PROGRAM P90_Interlock
VAR_INPUT
	bRecipeRunning 		: BOOL;
	RecipeStopped 		: BOOL;
	ManualOperation 	: BOOL;
	bInductionHeaterMC	: BOOL;
	bThermalBathMC		: BOOL;
	bVacuumPumpMC 		: BOOL;
	bLineHeaterMC 		: BOOL; 
END_VAR
VAR_OUTPUT
	bRecipeStartAvailable	: BOOL;
	bReactorOpenEnable		: BOOL;
	bHeaterOnEnable			: BOOL;
	bPumpOnEnable			: BOOL;
	
	bDorOnEnable			: BOOL;
	bDorOffEnable			: BOOL;
	bOpenEnableTemp			: BOOL;
	bOpenEnablePress		: BOOL;	
	
	bPowerResetSwitch		: BOOL;
	bMainPowerMonitor		: BOOL;

	AlarmTrig				: BOOL;
	WarningTrig				: BOOL;
	bMaintKey				: BOOL;
	bGasStateProcess		: BOOL;
	bGasStateSource			: BOOL;
	bGasStateVent			: BOOL;
END_VAR	
VAR
	bPowerResetLED			: BOOL;
	bUPSMode				: BOOL;
	tAlarmDelay_A			: TIME; //아날로그 디바이스 지연시간
	tAlarmDelay_D			: TIME; //디지털 디바이스 지연시간
	
	fbDeviationCheck		:ARRAY[1..29] OF FB_DeviationCheck;
	wDeviceAlarmEnable		: DWORD;
	wDeviceWarningEnable	: DWORD;
	bDeviationAlarm			: BOOL;
	bDeviationWarning		: BOOL;
	wDeviationAlarm			: DWORD;
	wDeviationWarning		: DWORD;

	fbSensorLimitCheck		:ARRAY[1..4] OF FB_SensorLimitCheck;
	wLimitAlarmEnable		: DWORD;
	wLimitWarningEnable		: DWORD;
	bLimitAlarm				: BOOL;
	bLimitWarning			: BOOL;
	wLimitAlarm				: DWORD;
	wLimitWarning			: DWORD;
	
	fbFaultCheck			:ARRAY[1..6] OF FB_FaultCheck;
	wAlarmEnable			: DWORD;
	wWarningEnable			: DWORD;

	bFaultAlarm				: BOOL;
	bFaultWarning			: BOOL;
	wAlarm					: DWORD;
	wWarning				: DWORD;
		
	bAlarmEnable			: BOOL;
	bWarningEnable			: BOOL;
	bDeviceCurrentAlarmState	: BOOL;
	bDeviceCurrentWarningState 	: BOOL;
	fDeviceCurrentValue			: REAL;
	fDeviceAlarmTreshold		: REAL;
	fDeviceWarningTreshold		: REAL;
	
	i	: INT;
	j 	: INT;
	
END_VAR

(* Read from Device*)
//Interlock Variable Set
bMaintKey := GVL_IO.aDigitalInputIO[1].0;
bPowerResetSwitch := GVL_IO.aDigitalInputIO[1].1;
bMainPowerMonitor := GVL_IO.aDigitalInputIO[7].5;
bGasStateProcess := GVL_IO.aOutputSolValve[1].0 AND //HYD Carrier Change Valve
	GVL_IO.aOutputSolValve[1].1 AND //Main Carrier Change Valve
	GVL_IO.aOutputSolValve[1].2 AND //SiH4 Source Change Valve
	GVL_IO.aOutputSolValve[1].3 //NH3 Source Change Valve
	; //All False이면 Safety State
bGasStateSource := GVL_IO.aOutputSolValve[1].4 AND GVL_IO.aOutputSolValve[1].5 AND GVL_IO.aOutputSolValve[1].6 AND //Source #1
	GVL_IO.aOutputSolValve[1].7 AND GVL_IO.aOutputSolValve[1].8 AND GVL_IO.aOutputSolValve[1].9 AND //Source #2
	GVL_IO.aOutputSolValve[1].10 AND GVL_IO.aOutputSolValve[1].11 AND GVL_IO.aOutputSolValve[1].12 AND //Source #3
	GVL_IO.aOutputSolValve[1].13 AND GVL_IO.aOutputSolValve[1].14 AND GVL_IO.aOutputSolValve[1].15 AND //Source #4
	GVL_IO.aOutputSolValve[2].0 AND GVL_IO.aOutputSolValve[2].1 AND GVL_IO.aOutputSolValve[2].2 AND //Source #5
	GVL_IO.aOutputSolValve[2].3 AND GVL_IO.aOutputSolValve[2].4 AND GVL_IO.aOutputSolValve[2].6 //Source #6
	; //All False이면 Safety State
bGasStateVent := GVL_IO.aOutputSolValve[2].15;
GVL_IO.aInterlock[1].10 := bRecipeStartAvailable;
GVL_IO.aInterlock[1].11 := bReactorOpenEnable;
GVL_IO.aInterlock[1].12 := bHeaterOnEnable;
GVL_IO.aInterlock[1].13 := bPumpOnEnable;

//Sinal Tower Set
IF (bMaintKey = TRUE) THEN //bMaintKey 변경
	P92_Maintenance.nCaseSignalTower		:= 5; //Signal Tower White - Maintenance
ELSIF (bMaintKey = FALSE) AND MAIN.bOperationMode = FALSE THEN
	P92_Maintenance.nCaseSignalTower		:= 4; //Signal Tower Blue - Idle
END_IF

//알람 지연 시간 변환
tAlarmDelay_A := REAL_TO_TIME(GVL_IO.aInterlockSet[3]*1000); // UI Setting Analog Delay Time Value(Miliseconde)
tAlarmDelay_D := REAL_TO_TIME(GVL_IO.aInterlockSet[4]*1000);

//Controller Deviation Monitoring - MFC/EPC
IF (bMaintKey = FALSE) THEN
	FOR i := 1 TO 26 DO
		wDeviceAlarmEnable := SHR(GVL_IO.aInterlockEnable[2], (i+2)); //오늘쪽 쉬프트 연산
		wDeviceWarningEnable := SHR(GVL_IO.aInterlockEnable[3], (i+2));
		fbDeviationCheck[i](
			bAlarmEnable := wDeviceAlarmEnable.0,
			bWarningEnable := wDeviceWarningEnable.0,
			fCurrentValue := GVL_IO.aController_PV[i],
			fControlValue := GVL_IO.aController_CV[i],
			fMaxValue := GVL_IO.aMaxValueController[i],
			fAlarmTreshold := GVL_IO.aInterlockSet[1],
			fWarningTreshold := GVL_IO.aInterlockSet[2],
			tAlarmDelay := tAlarmDelay_A,
			bDeviationAlarm => bDeviationAlarm, //알람 출력
			bDeviationWarning => bDeviationWarning // 주의(Warning) 출력
			);
		IF bDeviationAlarm THEN		
			GVL_IO.aInterlock[1].0 := TRUE; //Alarm Trig
			P92_Maintenance.nCaseSignalTower := 1; // Signal Tower RED - Alarm
			wDeviationAlarm := ROR(GVL_IO.aInterlock[3], (i+2));
			wDeviationAlarm.0 := TRUE;
			GVL_IO.aInterlock[3] := ROL(wDeviationAlarm, (i+2));
		ELSE
			wDeviationAlarm := ROR(GVL_IO.aInterlock[3], (i+2));
			wDeviationAlarm.0 := FALSE;
			GVL_IO.aInterlock[3] := ROL(wDeviationAlarm, (i+2));	
		END_IF
		
		IF bDeviationWarning THEN
			GVL_IO.aInterlock[1].1 := TRUE; // Warning Trig
			P92_Maintenance.nCaseSignalTower := 2; // Signal Tower Yellow - Warning
			wDeviationWarning := ROR(GVL_IO.aInterlock[5], (i+2));
			wDeviationWarning.0 := TRUE;
			GVL_IO.aInterlock[5] := ROL(wDeviationWarning, (i+2));
		ELSE
			wDeviationWarning := ROR(GVL_IO.aInterlock[5], (i+2));
			wDeviationWarning.0 := FALSE;
			GVL_IO.aInterlock[5] := ROL(wDeviationWarning, (i+2));
		END_IF
	END_FOR
	//Controller Deviation Monitoring - Temp, Pressure, Rotation
	FOR i := 27 TO 29 DO
		wDeviceAlarmEnable := SHR(GVL_IO.aInterlockEnable[2], (i-27)); //오늘쪽 쉬프트 연산, -27은 어레이 변수 옵셋값
		wDeviceWarningEnable := SHR(GVL_IO.aInterlockEnable[3], (i-27));
		fbDeviationCheck[i](
			bAlarmEnable := wDeviceAlarmEnable.0,
			bWarningEnable := wDeviceWarningEnable.0,
			fCurrentValue := GVL_IO.aController_PV[i],
			fControlValue := GVL_IO.aController_CV[i],
			fMaxValue := GVL_IO.aMaxValueController[i],
			fAlarmTreshold := GVL_IO.aInterlockSet[1],
			fWarningTreshold := GVL_IO.aInterlockSet[2],
			tAlarmDelay := tAlarmDelay_A,
			bDeviationAlarm => bDeviationAlarm, //알람 출력
			bDeviationWarning => bDeviationWarning // 주의(Warning) 출력
			);
		IF bDeviationAlarm THEN		
			GVL_IO.aInterlock[1].0 := TRUE; //Alarm Trig
			P92_Maintenance.nCaseSignalTower := 1; // Signal Tower RED - Alarm
			wDeviationAlarm := ROR(GVL_IO.aInterlock[3], (i-27));
			wDeviationAlarm.0 := TRUE;
			GVL_IO.aInterlock[3] := ROL(wDeviationAlarm, (i-27));
		ELSE
			wDeviationAlarm := ROR(GVL_IO.aInterlock[3], (i-27));
			wDeviationAlarm.0 := FALSE;
			GVL_IO.aInterlock[3] := ROL(wDeviationAlarm, (i-27));
		END_IF
		
		IF bDeviationWarning THEN
			GVL_IO.aInterlock[1].1 := TRUE; // Warning Trig
			P92_Maintenance.nCaseSignalTower := 2; // Signal Tower Yellow - Warning
			wDeviationWarning := ROR(GVL_IO.aInterlock[5], (i-27));
			wDeviationWarning.0 := TRUE;
			GVL_IO.aInterlock[5] := ROL(wDeviationWarning, (i-27));
		ELSE
			wDeviationWarning := ROR(GVL_IO.aInterlock[5], (i-27));
			wDeviationWarning.0 := FALSE;
			GVL_IO.aInterlock[5] := ROL(wDeviationWarning, (i-27));
		END_IF	
	END_FOR
	//Gas Pressure Alarm N2, H2, NH3, SiH4
	FOR i := 1 TO 4 DO
		wLimitAlarmEnable := SHR(GVL_IO.aInterlockEnable[4], (i-1)); //오늘쪽 쉬프트 연산, 은 어레이 변수 옵셋값
		wLimitWarningEnable := SHR(GVL_IO.aInterlockEnable[5], (i-1));
		fbSensorLimitCheck[i](
			bAlarmEnable := wLimitAlarmEnable.0,
			bWarningEnable := wLimitWarningEnable.0,
			fCurrentValue := GVL_IO.aMonitoring_PV[(i+3)],
			fAlarmTreshold := GVL_IO.aInterlockSet[5],
			fWarningTreshold := GVL_IO.aInterlockSet[6],
			tAlarmDelay := tAlarmDelay_D,
			bLimitAlarm => bLimitAlarm, //알람 출력
			bLimitWarning => bLimitWarning //주의(Warning) 출력
			);	
		IF bLimitAlarm THEN		
			GVL_IO.aInterlock[1].0 := TRUE; //Alarm Trig
			P92_Maintenance.nCaseSignalTower := 1; // Signal Tower RED - Alarm
			//팝업 표시
			wLimitAlarm := ROR(GVL_IO.aInterlock[2], (i-1));
			wLimitAlarm.0 := TRUE;
			GVL_IO.aInterlock[2] := ROL(wLimitAlarm, (i-1));
			//대시보드 표시
			wLimitAlarm := ROR(GVL_IO.aInterlock[1], (i*2));
			wLimitAlarm.0 := TRUE;
			GVL_IO.aInterlock[1] := ROL(wLimitAlarm, (i*2));
		ELSE
			//팝업 표시
			wLimitAlarm := ROR(GVL_IO.aInterlock[2], (i-1));
			wLimitAlarm.0 := FALSE;
			GVL_IO.aInterlock[2] := ROL(wLimitAlarm, (i-1));
			//대시보드 표시
			wLimitAlarm := ROR(GVL_IO.aInterlock[1], (i*2));
			wLimitAlarm.0 := FALSE;
			GVL_IO.aInterlock[1] := ROL(wLimitAlarm, (i*2));
		END_IF
		
		IF bLimitWarning THEN		
			GVL_IO.aInterlock[1].1 := TRUE; //Warning Trig
			P92_Maintenance.nCaseSignalTower := 2; // Signal Tower YELLOW - Warning
			//팝업 표시
			wLimitWarning := ROR(GVL_IO.aInterlock[4], (i-1));
			wLimitWarning.0 := TRUE;
			GVL_IO.aInterlock[4] := ROL(wLimitWarning, (i-1));
			//대시보드 표시
			wLimitWarning := ROR(GVL_IO.aInterlock[1], (i*2)+1);
			wLimitWarning.0 := TRUE;
			GVL_IO.aInterlock[1] := ROL(wLimitWarning, (i*2)+1);
		ELSE
			//팝업 표시
			wLimitWarning := ROR(GVL_IO.aInterlock[4], (i-1));
			wLimitWarning.0 := FALSE;
			GVL_IO.aInterlock[4] := ROL(wLimitWarning, (i-1));
			//대시보드 표시
			wLimitWarning := ROR(GVL_IO.aInterlock[1], (i*2)+1);
			wLimitWarning.0 := FALSE;
			GVL_IO.aInterlock[1] := ROL(wLimitWarning, (i*2)+1);
		END_IF
	END_FOR
	
	//Cooling Water Over Temperature, Susceptor Over Temperature, Reactor Over Pressure
	FOR i := 1 TO 4 DO
		CASE i OF
			1: //CW Temperature High S/H
				bAlarmEnable := GVL_IO.aInterlockEnable[4].4;
				bWarningEnable := GVL_IO.aInterlockEnable[5].4;
				fDeviceCurrentValue := GVL_IO.aMonitoring_PV[8];
				fDeviceAlarmTreshold := GVL_IO.aInterlockSet[7];
				fDeviceWarningTreshold := GVL_IO.aInterlockSet[8];
			2: //CW Temperature High Coil
				bAlarmEnable := GVL_IO.aInterlockEnable[4].5;
				bWarningEnable := GVL_IO.aInterlockEnable[5].5;
				fDeviceCurrentValue := GVL_IO.aMonitoring_PV[9];
				fDeviceAlarmTreshold := GVL_IO.aInterlockSet[9];
				fDeviceWarningTreshold := GVL_IO.aInterlockSet[10];
			3: //Susceptor Over Temperature
				bAlarmEnable := GVL_IO.aInterlockEnable[4].6;
				bWarningEnable := GVL_IO.aInterlockEnable[5].6;
				fDeviceCurrentValue := GVL_IO.aController_PV[27];
				fDeviceAlarmTreshold := GVL_IO.aInterlockSet[11];
				fDeviceWarningTreshold := (GVL_IO.aInterlockSet[11] - 20.0); //20도 아래에서 Warning 발생				
			4: //Reactor Over Pressure Alarm
				bAlarmEnable := GVL_IO.aInterlockEnable[4].7;
				bWarningEnable := GVL_IO.aInterlockEnable[5].7;
				fDeviceCurrentValue := GVL_IO.aController_PV[28];
				fDeviceAlarmTreshold := GVL_IO.aInterlockSet[12];
				fDeviceWarningTreshold := (GVL_IO.aInterlockSet[12] - 50.0); //50Torr 아래에서 Warning 발생							
		END_CASE
		fbSensorLimitCheck[i](
			bAlarmEnable := bAlarmEnable,
			bWarningEnable := bWarningEnable,
			fCurrentValue := fDeviceCurrentValue,
			fAlarmTreshold := fDeviceAlarmTreshold,
			fWarningTreshold := fDeviceWarningTreshold,
			tAlarmDelay := tAlarmDelay_D,
			bLimitAlarm => bLimitAlarm, //알람 출력
			bLimitWarning => bLimitWarning //주의(Warning) 출력
			);
		IF bLimitAlarm THEN		
			GVL_IO.aInterlock[1].0 := TRUE; //Alarm Trig
			P92_Maintenance.nCaseSignalTower := 1; // Signal Tower RED - Alarm
			wDeviationAlarm := ROR(GVL_IO.aInterlock[2], (i+3));
			wDeviationAlarm.0 := TRUE;
			GVL_IO.aInterlock[2] := ROL(wDeviationAlarm, (i+3));
		ELSE
			wDeviationAlarm := ROR(GVL_IO.aInterlock[2], (i+3));
			wDeviationAlarm.0 := FALSE;
			GVL_IO.aInterlock[2] := ROL(wDeviationAlarm, (i+3));
		END_IF
		
		IF bDeviationWarning THEN
			GVL_IO.aInterlock[1].1 := TRUE; // Warning Trig
			P92_Maintenance.nCaseSignalTower := 2; // Signal Tower Yellow - Warning
			wDeviationWarning := ROR(GVL_IO.aInterlock[4], (i+3));
			wDeviationWarning.0 := TRUE;
			GVL_IO.aInterlock[4] := ROL(wDeviationWarning, (i+3));
		ELSE
			wDeviationWarning := ROR(GVL_IO.aInterlock[4], (i+3));
			wDeviationWarning.0 := FALSE;
			GVL_IO.aInterlock[4] := ROL(wDeviationWarning, (i+3));
		END_IF		
	END_FOR
	
	//Device Fault Check - Pneumatic, Heater, Pump, Motor, GC Door, RC Door
	FOR i := 1 TO 8 DO
		CASE i OF
			1: //CDA Alarm Switch (Pneumatic)
				bAlarmEnable := GVL_IO.aInterlockEnable[4].8;
				bWarningEnable := GVL_IO.aInterlockEnable[5].8;
				bDeviceCurrentAlarmState := GVL_IO.aInputState[1].4;
				bDeviceCurrentWarningState := GVL_IO.aInputState[1].4;
			2: //Cooling Water Switch
				bAlarmEnable := GVL_IO.aInterlockEnable[4].9;
				bWarningEnable := GVL_IO.aInterlockEnable[5].9;
				bDeviceCurrentAlarmState := GVL_IO.aInputState[1].5;
				bDeviceCurrentWarningState := GVL_IO.aInputState[1].5;
			3: //Induction Heater Fault
				bAlarmEnable := GVL_IO.aInterlockEnable[4].10;
				bWarningEnable := GVL_IO.aInterlockEnable[5].10;
				bDeviceCurrentAlarmState := GVL_IO.aInputState[1].8;
				bDeviceCurrentWarningState := GVL_IO.aInputState[1].8;
			4: //Rotatin Motor Fault
				bAlarmEnable := GVL_IO.aInterlockEnable[4].11;
				bWarningEnable := GVL_IO.aInterlockEnable[5].11;
				bDeviceCurrentAlarmState := GVL_IO.aInputState[1].11;
				bDeviceCurrentWarningState := GVL_IO.aInputState[1].11;
			5: //Vacuum Pump Fault
				bAlarmEnable := GVL_IO.aInterlockEnable[4].12;
				bWarningEnable := GVL_IO.aInterlockEnable[5].12;
				bDeviceCurrentAlarmState := GVL_IO.aInputState[1].12;
				bDeviceCurrentWarningState := GVL_IO.aInputState[1].14;
			6: //Gas Cabinet Door Open
				bAlarmEnable := GVL_IO.aInterlockEnable[4].13;
				bWarningEnable := GVL_IO.aInterlockEnable[5].13;
				bDeviceCurrentAlarmState := GVL_IO.aInputState[2].0;
				bDeviceCurrentWarningState := GVL_IO.aInputState[2].0;
			7: //Reactor Cabinet Door Open
				bAlarmEnable := GVL_IO.aInterlockEnable[4].14;
				bWarningEnable := GVL_IO.aInterlockEnable[5].14;
				bDeviceCurrentAlarmState := GVL_IO.aInputState[2].1;
				bDeviceCurrentWarningState := GVL_IO.aInputState[2].1;
			8: //DOR Fault
				bAlarmEnable := GVL_IO.aInterlockEnable[4].15;
				bWarningEnable := GVL_IO.aInterlockEnable[5].15;
				IF (P17_DOROperation.bError = 1) THEN
					bDeviceCurrentAlarmState := TRUE;
				ELSE
					bDeviceCurrentAlarmState := FALSE;
				END_IF
				IF (P17_DOROperation.bError = 2) OR (P17_DOROperation.bError = 3) THEN
					bDeviceCurrentWarningState := TRUE;
				ELSE
					bDeviceCurrentWarningState := FALSE;
				END_IF
		END_CASE

		fbFaultCheck[i](
			bAlarmEnable := bAlarmEnable,
			bWarningEnable := bWarningEnable,
			bCurrentAlarmState := bDeviceCurrentAlarmState,
			bCurrentWarningState := bDeviceCurrentWarningState,
			tAlarmDelay := tAlarmDelay_D,
			bAlarm => bFaultAlarm,
			bWarning => bFaultWarning
			);
			
		IF bFaultAlarm THEN
			GVL_IO.aInterlock[1].0 := TRUE; //Alarm Trig
			P92_Maintenance.nCaseSignalTower := 1; // Signal Tower RED - Alarm
			//팝업 표시
			wAlarm := ROR(GVL_IO.aInterlock[2], (i+7));
			wAlarm.0 := TRUE;
			GVL_IO.aInterlock[2] := ROL(wAlarm, (i+7));
		END_IF
		IF bFaultWarning THEN
			GVL_IO.aInterlock[1].1 := TRUE; //Warning Trig
			P92_Maintenance.nCaseSignalTower := 2; // Signal Tower YELLOW - Warning
			//팝업 표시
			wAlarm := ROR(GVL_IO.aInterlock[4], (i+7));
			wAlarm.0 := TRUE;
			GVL_IO.aInterlock[4] := ROL(wAlarm, (i+7));
		END_IF
	END_FOR
	
	IF GVL_IO.aInterlockEnable[1].0 THEN //알람 리셋 버턴을 눌렀을 때
		GVL_IO.aInterlock[1].0 := FALSE; //Alarm Trig Reset
		GVL_IO.aInterlockEnable[1].0 := FALSE; //버턴 초기화
		P92_Maintenance.nCaseSignalTower := 4; // Signal Tower Blue - Idle
	END_IF
	IF GVL_IO.aInterlockEnable[1].1 THEN //주의 리셋 버턴을 눌렀을 때
		GVL_IO.aInterlock[1].1 := FALSE; //Warmomg Trig Reset
		GVL_IO.aInterlockEnable[1].1 := FALSE; //버턴 초기화
		P92_Maintenance.nCaseSignalTower := 4; // Signal Tower Blue - Idle
	END_IF	
ELSE
	//매인터넌스 키가 ON 되었을 때 MC(Induction, Bath, Pump, L_Heater) 조작 허용
	P92_Maintenance.nCaseSignalTower := 4; // Signal Tower Blue - Idle
	GVL_IO.aDigitalOutputIO[3].0 := bInductionHeaterMC;
	GVL_IO.aDigitalOutputIO[3].1 := bThermalBathMC;
	GVL_IO.aDigitalOutputIO[3].2 := bVacuumPumpMC;
	GVL_IO.aDigitalOutputIO[3].3 := bLineHeaterMC;
END_IF

bRecipeStartAvailable := //레시피 가능한 상태이면 TRUE
	NOT(AlarmTrig) AND
	NOT(WarningTrig) AND
	NOT(bMaintKey) AND
	GVL_IO.aInputState[2].4 AND //Cover Lower Limt
	GVL_IO.aInputState[4].6 AND //DOR State
	NOT(RCP.state_RcpOperation = 10) AND //Not Recipe Run State
	NOT(bGasStateProcess) AND //Safety Process Gas : TRUE
	NOT(bGasStateSource) AND //Safety Source Gas : TRUE
	NOT(bGasStateVent) AND
	P11_E3508. bManAuto_E3508 AND //Temperature Controller Auto : True
	P12_IQ_PLUS. ingPressureControl //Throttle Valve Pressure Control Mode : True 
	;

bDorOnEnable :=
	NOT(AlarmTrig) AND
	P16_CoverOperation.isCoverClosed AND
	P17_DOROperation.isDOROnState AND
	P12_IQ_PLUS.isPumpRunning
	;
bHeaterOnEnable := bDorOnEnable;

// DOR Off Conditions
IF  GVL_IO.aController_PV[27] < GVL_IO.aInterlockSet[13] THEN
	bOpenEnableTemp := TRUE;
ELSE
	bOpenEnableTemp := FALSE;
END_IF
IF  GVL_IO.aController_PV[28] < GVL_IO.aInterlockSet[14] THEN
	bOpenEnablePress := TRUE;
ELSE
	bOpenEnablePress := FALSE;
END_IF
bDorOffEnable :=
	NOT(AlarmTrig) AND
	NOT(P17_DOROperation.isDOROnState) AND
	NOT(RCP.state_RcpOperation = 10) AND //Not Recipe Run State
	NOT(bGasStateProcess) AND //Safety Process Gas : TRUE
	NOT(bGasStateSource) AND //Safety Source Gas : TRUE
	bGasStateVent AND //Vent Valve는 펌프 뒤쪽 Open
	NOT(GVL_IO.aInterlockEnable[6].4) AND //Can Open Temperature Check
	bOpenEnableTemp AND
	NOT(GVL_IO.aInterlockEnable[6].5) AND //Can Open Pressure Check
	bOpenEnablePress ;
	;
bReactorOpenEnable := bDorOffEnable;

(* Out to Device*)
GVL_IO.aDigitalOutputIO[3].7 := bPowerResetLED;
GVL_IO.aDigitalOutputIO[2].4 := bUPSMode;

END_PROGRAM

(* stored: Version 1.1.0.1, ProductVersion 3.1.4026.11
   POU P90_Interlock: Id {c8b81d81-de46-4c7a-a894-4387b2cd9bf7}, SpecialFunc None *)
